TYPE ST_CoaxVisionResult :
STRUCT
    // TRUE仅表示真实测量或Simulation结果有效；Fallback时保持FALSE。
    bValid      : BOOL;
    fCoaxiality : LREAL;
    fDeltaX     : LREAL;
    fDeltaY     : LREAL;
    fCorrectionX : LREAL; // AdjustmentX mechanical relative correction, mm.
    fCorrectionY : LREAL; // AdjustmentY mechanical relative correction, mm.
END_STRUCT
END_TYPE

(* stored: Version 1.1.0.1, ProductVersion 3.1.4026.20
   DUT ST_CoaxVisionResult: Id {1BD94FBF-BEB1-4A36-BBCB-6950A87F8FEC} *)
